TYPE Read_AR_Values_To_PC_Struct :
UNION
	S_ARValues_To_PC:S_ARValues_To_PC_Struct;
END_UNION
END_TYPE

(* stored: Version 1.1.0.1, ProductVersion 3.1.4024.16
   DUT Read_AR_Values_To_PC_Struct: Id {f78d6820-244b-4cb1-8ac4-103579545187} *)
